TYPE SC_SENSOR_BeltConveyors :
(
	eCounterSensor := 1,
	eBeltConveyorsMaxSensors
)UINT;
END_TYPE

(* stored: Version 1.1.0.1, ProductVersion 3.1.4024.2
   DUT SC_SENSOR_BeltConveyors: Id {9b6b561d-f00f-48b3-872c-2f3bd12b6eb7} *)
